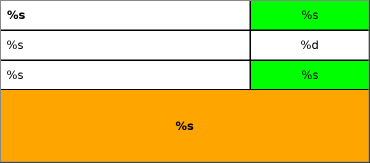
VISUALIZATION VISU_MODE_QUARTZ  // 370x163
VAR_INPUT
	m_input_Mode_Quartz:		BLOCK_1RUN_1QUARTZ;
END_VAR
    Rectangle (0,0 250x30), "%s", text list: 'TextList_1Run_1Quartz', text index: 0
    Rectangle (0,30 250x30), "%s", invisible if: not m_input_Mode_Quartz.STATE_Mode, text list: 'TextList_1Run_1Quartz', text index: 4
    Rectangle (0,60 250x30), "%s", text list: 'TextList_1Run_1Quartz', text index: 3
    Rectangle (250,0 120x30), "%s", colour toggle: MACHINE.CONF_Standby_Auto, invisible if: m_input_Mode_Quartz.STATE_Mode, text list: 'TextList_1Run_1Quartz', text index: 2
    Rectangle (250,0 120x30), "%s", colour toggle: MACHINE.CONF_Standby_Auto, invisible if: not m_input_Mode_Quartz.STATE_Mode, text list: 'TextList_1Run_1Quartz', text index: 1
    Rectangle (250,60 120x30), "%s", colour toggle: MACHINE.CONF_Standby_Auto, invisible if: m_input_Mode_Quartz.STATE_RAZ_Quartz, text list: 'TextList_1Run_1Quartz', text index: 2
    Rectangle (250,60 120x30), "%s", colour toggle: MACHINE.CONF_Standby_Auto, invisible if: not m_input_Mode_Quartz.STATE_RAZ_Quartz, text list: 'TextList_1Run_1Quartz', text index: 1
    Rectangle (250,30 120x30), "%d", text variable: m_input_Mode_Quartz.STATE_Next_Quartz, invisible if: not m_input_Mode_Quartz.STATE_Mode
    Rectangle (0,89 370x74), "%s", invisible if: not m_input_Mode_Quartz.RQ_Disp_Change_Quartz, text list: 'TextList_1Run_1Quartz', text index: 5
    Rectangle (250,0 120x30), colour toggle: MACHINE.CONF_Standby_Auto, invisible if: MODE_QUARTZ_PROD.I_Prod
        tap MODE_QUARTZ_PROD.M_Mode
    Rectangle (250,59 120x30), colour toggle: MACHINE.CONF_Standby_Auto, invisible if: not MODE_QUARTZ_PROD.STATE_Mode
        tap MODE_QUARTZ_PROD.M_RAZ_Quartz
END_VISUALIZATION

(* stored: Version 1.1.0.1, ProductVersion 3.1.4024.12
   Visu VISU_MODE_QUARTZ: Id {c953bcc6-96e3-47f7-88c9-46fa5ad55a58} *)
